FUNCTION_BLOCK SAE_J1939_WORD_TO_PERCENT (* convert a hexadecimal Percent to a REAL *)
  (* Standard: 61499-2; Description: Copyright (c) 2023 HR Agrartechnik GmbH This program and the accompanying materials are made available under the terms of the Eclipse Public License 2.0 which is available at https://www.eclipse.org/legal/epl-2.0/ SPDX-License-Identifier: EPL-2.0 Input should be a hexadecimal Type, mostly coming from a Fieldbus like SAE J1939 or ISO 11783 or similar. 0 % = 0x0 100 % = 0xFAFF all other Input Values should be ignored. so e.g. 0xFFFF will not change the Output Value. *)
  (* Version 1.0, 2023-06-06, Franz Höpfinger, HR Agrartechnik GmbH *)
  PACKAGE signalprocessing;
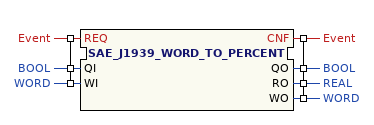
  EVENT_INPUT
    REQ WITH QI, WI; (* Service Request *)
  END_EVENT
  EVENT_OUTPUT
    CNF WITH QO, RO, WO; (* Confirmation of Requested Service *)
  END_EVENT
  VAR_INPUT
    QI : BOOL; (* Event Input Qualifier *)
    WI : WORD; (* 2-byte Data (16 bits) Input Value *)
  END_VAR
  VAR_OUTPUT
    QO : BOOL; (* Event Output Qualifier *)
    RO : REAL; (* Output in Percent as REAL *)
    WO : WORD; (* Raw data Filtered to 0x0 .. 0xFAFF *)
  END_VAR
  VAR CONSTANT
    ISO_VALID_SIGNAL_W : WORD := 16#FAFF; (* 16 bit max value of valid signal; from SAE J1939 *)
  END_VAR
  ALGORITHM REQ IN ST:
QO := QI;
IF (TRUE = QI) THEN
	IF (WI <= ISO_VALID_SIGNAL_W) THEN
		WO := WI;
		RO := UDINT_TO_REAL(WORD_TO_UDINT(WO)) / UDINT_TO_REAL(WORD_TO_UDINT(ISO_VALID_SIGNAL_W));
	END_IF;
END_IF;
  END_ALGORITHM
END_FUNCTION_BLOCK
